// TwinCAT 3 PLC project TestProj
// ProgramVersion: 3.1.4022.7
// libraries:
//   Tc2_Standard, * (Beckhoff Automation GmbH)
//   Tc2_System, * (Beckhoff Automation GmbH)
//   Tc2_Utilities, * (Beckhoff Automation GmbH)
//   Tc3_Module, * (Beckhoff Automation GmbH)
//   Tc3_RealtimeMonitoring, * (Beckhoff Automation GmbH)
// project tree:
//   DUTs/ TestStruct.TcDUT
//   / PlcTask.TcTTO
//   POUs/ MAIN.TcPOU
// real-time tasks:
//   TASK PlcTask: cycle T#10ms, priority 20, ADS port 350

CONFIGURATION TestProj
    RESOURCE PLC ON TwinCAT3
        TASK PlcTask(INTERVAL := T#10ms, PRIORITY := 20);
        PROGRAM MAIN WITH PlcTask : MAIN;
    END_RESOURCE
END_CONFIGURATION

// ---- DUTs/TestStruct.TcDUT
TYPE TestStruct :
STRUCT
    {attribute 'pytmc' := '
        pv: Number
        io: i
     '}
    Number : LREAL;
    {attribute 'pytmc' := '
        pv: OK
        io: i
     '}
    Bin : BOOL;
END_STRUCT
END_TYPE

// ---- POUs/MAIN.TcPOU
PROGRAM MAIN
VAR CONSTANT
    TestSize : INT := 5000;
END_VAR
VAR
    {attribute 'pytmc' := '
        pv: TestArray
     '}
    TestArray : ARRAY [0..TestSize] OF TestStruct;
    NoiseRand : DRAND := (Seed:=0);
    idx : INT;
    firstpass : BOOL := TRUE;
    {attribute 'pytmc' := '
        pv: LastExecTime
        io: i
     '}
    LastExecTime : UDINT;
    CycleTime : UDINT;
    fbGetCurTaskIdx  : GETCURTASKINDEX;
    
    fbRTM : FB_RTMon_LogMark;
    
    fbRouterStatus : FB_GetRouterStatusInfo;
    RouterInfo : ST_TcRouterStatusInfo;
END_VAR

fbRTM.LogIntervalStart(1,1);

fbRTM.LogSequenceStart(1,2);
For idx := 0 to TestSize DO
    NoiseRand();
    TestArray[idx].Number := NoiseRand.Num;
    TestArray[idx].Bin := NoiseRand.Num > 0.5;
END_FOR
fbRTM.LogSequenceStop(1,2);

IF firstpass THEN 
    fbGetCurTaskIdx();
    firstpass := false;
END_IF
LastExecTime := _TaskInfo[fbGetCurTaskIdx.index].LastExecTime;

fbRTM.LogIntervalStop(1,1);

fbRouterStatus.bExecute S= NOT fbRouterStatus.bBusy;
fbRouterStatus.bExecute R= fbRouterStatus.bBusy;
fbRouterStatus();
IF NOT fbRouterStatus.bBusy THEN RouterInfo := fbRouterStatus.info; END_IF

END_PROGRAM
